FUNCTION Convert_TOD_TO_LINT : Hresult
VAR_INPUT
	in : TOD;
	out : REFERENCE TO LINT;
END_VAR
VAR
	converted : LINT;
END_VAR

converted := TOD_TO_LINT(in);

IF (LINT_TO_TOD(converted) <> in) THEN
	Convert_TOD_TO_LINT := INCOMPATIBLE;
	RETURN;
END_IF

out := converted;

END_FUNCTION

(* stored: Version 1.1.0.1, ProductVersion 3.1.4024.12
   POU Convert_TOD_TO_LINT: Id {9539b7b6-653e-441d-b901-21c33bbb7c84}, SpecialFunc None *)
